// TIA Portal V18 export
FUNCTION_BLOCK "myFunctionBlock"   // FB2, LAD
{ S7_Optimized_Access := 'TRUE' }
VERSION : 0.1
// stored: AutoNumber true, IsIECCheckEnabled false, IsRetainMemResEnabled false, MemoryReserve 100, SetENOAutomatically false, UDAEnableTagReadback false
   VAR_OUTPUT
      Lamp : Bool;
   END_VAR
   VAR
      Start : Bool;
      Stop : Bool;
   END_VAR
BEGIN

REGION Network 1
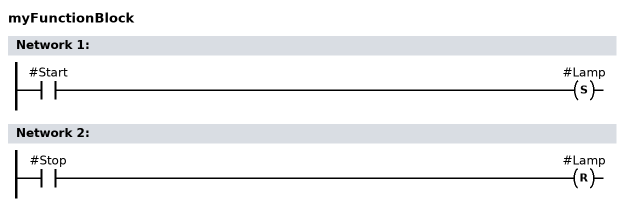
   RUNG wire#powerrail
      Contact( #Start )
      S_Coil( #Lamp )
   END_RUNG
   // the same network as SCL:
   IF #Start THEN #Lamp := TRUE; END_IF;
END_REGION

REGION Network 2
   RUNG wire#powerrail
      Contact( #Stop )
      R_Coil( #Lamp )
   END_RUNG
   // the same network as SCL:
   IF #Stop THEN #Lamp := FALSE; END_IF;
END_REGION
END_FUNCTION_BLOCK
